
FUNCTION CB_sint_to_bool : BOOL


TITLE = ' Convert an integer into a boolean '
VERSION : '1.0'
AUTHOR  : CB
NAME    : sintToBo
FAMILY  : TNI

VAR_INPUT
    IN : INT;
END_VAR

BEGIN

CB_sint_to_bool := (IN <>0);

END_FUNCTION
